PROGRAM prgEM
VAR
		// Grid Objekt H 3-phase, 400V
//	fb_UV_Garderobe					: FB_Shelly_3EM;
	fb_UV_Garderobe					: FB_Shelly_Pro3EM;
	
	lrPower_UV_Garderobe_TotalkW		: LREAL;			//{#lynus.ag#()}
	lrEnergy_UV_Garderobe_Total			: LREAL;			//{#lynus.ag#()}
	lrCurrent_UV_Garderobe_L1			: LREAL;			//{#lynus.ag#()}
	lrCurrent_UV_Garderobe_L2			: LREAL;			//{#lynus.ag#()}
	lrCurrent_UV_Garderobe_L3			: LREAL;			//{#lynus.ag#()}
	lrVoltage_UV_Garderobe_L1			: LREAL;			//{#lynus.ag#()}
	lrVoltage_UV_Garderobe_L2			: LREAL;			//{#lynus.ag#()}
	lrVoltage_UV_Garderobe_L3			: LREAL;			//{#lynus.ag#()}


	fb_Temperature_1				: FB_Shelly_hT;
	fb_Temperature_2				: FB_Shelly_HTplus;

	str_ip: STRING(15):='172.32.12.127';
	m_Start1: BOOL;
	m_Start2: BOOL;
	lrTemp1: LREAL;
	lrTemp2: LREAL;
END_VAR

	// Grid Objekt H 3-phase, 400V
(*
fb_UV_Garderobe(
	bStart:= , 
	tDelayRequest:= T#20S, 
	sHostname:= '172.32.12.121', 
	bValidResult=> , 
	bBusy=> , 
	bError=> , 
	bDone=> , 
	hrErrorCode=> ,
	lrtotalpower=> ,
	lrpowerL1=> ,
	lrpowerL2=> ,
	lrpowerL3=> ,
	lrcurrentL1=> lrCurrent_UV_Garderobe_L1,
	lrcurrentL2=> lrCurrent_UV_Garderobe_L2,
	lrcurrentL3=> lrCurrent_UV_Garderobe_L3,
	lrvoltageL1=> lrVoltage_UV_Garderobe_L1,
	lrvoltageL2=> lrVoltage_UV_Garderobe_L2,
	lrvoltageL3=> lrVoltage_UV_Garderobe_L3,
	lrenergyL1=> ,
	lrenergyL2=> ,
	lrenergyL3=>  );

lrPower_UV_Garderobe_TotalkW := 	fb_UV_Garderobe.lrtotalpower / 1000;
// sum-up energy
lrEnergy_UV_Garderobe_Total :=  fb_UV_Garderobe.lrenergyL1 + fb_UV_Garderobe.lrenergyL2 + fb_UV_Garderobe.lrenergyL3;
*)

fb_UV_Garderobe(
	bStart:= , 
	tDelayRequest:= T#20S, 
	sHostname:= '172.32.12.121', 
	bValidResult=> , );



fb_Temperature_1(
	bStart:= m_Start1, 
	tDelayRequest:= T#10S, 
	sHostname:= '172.32.12.127', 
	bValidResult=> , 
	bBusy=> , 
	bError=> , 
	bDone=> , 
	bConnected=> , 
	lr_Temperature=> , 
	lr_Humidity=> , 
	hrErrorCode=> );
	


fb_Temperature_2(
	bStart:= m_Start2, 
	tDelayRequest:= T#10S, 
	sHostname:= '172.32.12.124', 
	bValidResult=> , 
	bBusy=> , 
	bError=> , 
	bDone=> , 
	bConnected=> , 
	lr_Temperature=> , 
	lr_Humidity=> , 
	hrErrorCode=> );
	
IF fb_Temperature_1.lr_Temperature <> 0  THEN 
	lrTemp1 :=  fb_Temperature_1.lr_Temperature;
END_IF
IF fb_Temperature_2.lr_Temperature<>0 THEN
	lrTemp2 :=  fb_Temperature_2.lr_Temperature;
END_IF

END_PROGRAM

(* stored: Version 1.1.0.1, ProductVersion 3.1.4024.15
   POU prgEM: Id {3af41ed4-b9b9-451d-86e6-0d7631ab8bb0}, SpecialFunc None *)
